(******************************************************************************
Baustein: FB_TestBase
Spezifikation: doc/Spezifikation.pdf, Kap. x.y.z
-------------------------------------------------------------------------------
erstellt:
von:
Geändert:
von:
-------------------------------------------------------------------------------
Beschreibung
Dieser Baustein stellt die Basis für einen Unittest dar und enthält
alle notwendigen Variablen und Methoden zur Testauswertung.

-------------------------------------------------------------------------------
Input
-

Output
	o_eState : EState_t;
	o_eResult: EResult_t;
******************************************************************************)
FUNCTION_BLOCK FB_Assertion
VAR_OUTPUT
    o_eState    : EAssertion_t;
    o_u32Passed : UDINT;
    o_u32Failed : UDINT;
END_VAR

(******************************************************************************
Baustein: FB_TestBase.assertFALSE
Spezifikation: doc/Spezifikation.pdf, Kap. x.y.z
-------------------------------------------------------------------------------
erstellt:
von:
Geändert:
von:
-------------------------------------------------------------------------------
Beschreibung
Diese Methode...

-------------------------------------------------------------------------------
Input
	bValue : BOOL;

Output
-
******************************************************************************)
METHOD PROTECTED FINAL _FALSE : BOOL
VAR_INPUT
	bValue : BOOL;
END_VAR

	IF bValue = FALSE THEN
		addPassed();
	ELSE
		addFailed(bFatal := FALSE);
	END_IF
END_METHOD

(******************************************************************************
Baustein: FB_TestBase.assertFALSE_Fatal
Spezifikation: doc/Spezifikation.pdf, Kap. x.y.z
-------------------------------------------------------------------------------
erstellt:
von:
Geändert:
von:
-------------------------------------------------------------------------------
Beschreibung
Diese Methode

-------------------------------------------------------------------------------
Input
	bValue : BOOL;

Output
-
******************************************************************************)
METHOD PROTECTED FINAL _FALSE_Fatal : BOOL
VAR_INPUT
	bValue : BOOL;
END_VAR

	IF bValue = FALSE THEN
		addPassed();
	ELSE
		addFailed(bFatal := true);
	END_IF
END_METHOD

(******************************************************************************
Baustein: FB_TestBase.assertTRUE
Spezifikation: doc/Spezifikation.pdf, Kap. x.y.z
-------------------------------------------------------------------------------
erstellt:
von:
Geändert:
von:
-------------------------------------------------------------------------------
Beschreibung
Diese Methode...

-------------------------------------------------------------------------------
Input
	bValue : BOOL;

Output
-
******************************************************************************)
METHOD PROTECTED FINAL _TRUE : BOOL
VAR_INPUT
	bValue : BOOL;
END_VAR

	IF bValue = true THEN
		addPassed();
	ELSE
		addFailed(bFatal := FALSE);
	END_IF
END_METHOD


(******************************************************************************
Baustein: FB_TestBase.assertTRUE_Fatal
Spezifikation: doc/Spezifikation.pdf, Kap. x.y.z
-------------------------------------------------------------------------------
erstellt:
von:
Geändert:
von:
-------------------------------------------------------------------------------
Beschreibung
Diese Methode

-------------------------------------------------------------------------------
Input
-

Output
-
******************************************************************************)
METHOD PROTECTED FINAL _TRUE_Fatal : BOOL
VAR_INPUT
	bValue : BOOL;
END_VAR

	IF bValue = TRUE THEN
		addPassed();
	ELSE
		addFailed(bFatal := true);
	END_IF
END_METHOD

METHOD INTERNAL FINAL addFailed : BOOL
VAR_INPUT
    bFatal : BOOL;
END_VAR
	
    o_u32Failed := o_u32Failed + 1;
	
	o_eState := EAssertion_t.eStateFailed;
	
	IF bFatal = true THEN
		o_eState := EAssertion_t.eStateFailedFatal;
	END_IF
END_METHOD

METHOD INTERNAL FINAL addPassed : BOOL
	
    o_u32Passed := o_u32Passed + 1;
END_METHOD

(******************************************************************************
Baustein: FB_TestBase.assertEQUAL
Spezifikation: doc/Spezifikation.pdf, Kap. x.y.z
-------------------------------------------------------------------------------
erstellt:
von:
Geändert:
von:
-------------------------------------------------------------------------------
Beschreibung
Diese Methode

-------------------------------------------------------------------------------
Input
	Actual   : ANY;
	Expected : ANY;

Output
-
******************************************************************************)
METHOD PUBLIC FINAL EQUAL : BOOL
VAR_INPUT
	Actual   : ANY;
	Expected : ANY;
END_VAR
	EQUAL := FALSE;
	
	IF validate(Actual, Expected) = FALSE THEN
		addFailed(true);
		RETURN;
	END_IF
	
	_TRUE(MEMCMP(Actual.pValue, Expected.pValue, TO_UDINT(Actual.diSize)) = 0);
END_METHOD

(******************************************************************************
Baustein: FB_TestBase.assertEQUAL_Fatal
Spezifikation: doc/Spezifikation.pdf, Kap. x.y.z
-------------------------------------------------------------------------------
erstellt:
von:
Geändert:
von:
-------------------------------------------------------------------------------
Beschreibung
Diese Methode

-------------------------------------------------------------------------------
Input
	Actual   : ANY;
	Expected : ANY;

Output
-
******************************************************************************)
METHOD PUBLIC FINAL EQUAL_Fatal : BOOL
VAR_INPUT
	Actual   : ANY;
	Expected : ANY;
END_VAR
	EQUAL_Fatal := FALSE;
	
	IF validate(Actual, Expected) = FALSE THEN
		addFailed(true);
		RETURN;
	END_IF

	_TRUE_Fatal(MEMCMP(Actual.pValue, Expected.pValue, TO_UDINT(Actual.diSize)) = 0);
END_METHOD

(******************************************************************************
Baustein: FB_TestBase.logError
Spezifikation: doc/Spezifikation.pdf, Kap. x.y.z
-------------------------------------------------------------------------------
erstellt:
von:
Geändert:
von:
-------------------------------------------------------------------------------
Beschreibung
Diese Methode

-------------------------------------------------------------------------------
Input
-

Output
-
******************************************************************************)
{attribute 'hide'} 
METHOD PROTECTED FINAL logError : BOOL
VAR_INPUT
	i_strMessage : StrMessage_t;
END_VAR

	ADSLOGSTR(msgCtrlMask 	:= ADSLOG_MSGTYPE_ERROR , 
			  msgFmtStr 	:= i_strMessage, 
			  strArg 		:= '');
END_METHOD

(******************************************************************************
Baustein: FB_TestBase.assertNotEqual
Spezifikation: doc/Spezifikation.pdf, Kap. x.y.z
-------------------------------------------------------------------------------
erstellt:
von:
Geändert:
von:
-------------------------------------------------------------------------------
Beschreibung
Diese Methode

-------------------------------------------------------------------------------
Input
	Actual   : ANY;
	Expected : ANY;

Output
-
******************************************************************************)
METHOD PUBLIC FINAL NotEqual : BOOL
VAR_INPUT
	Actual   : ANY;
	Expected : ANY;
END_VAR
	NotEqual := FALSE;
	
	IF validate(Actual, Expected) = FALSE THEN
		addFailed(true);
		RETURN;
	END_IF
	
	_TRUE(MEMCMP(Actual.pValue, Expected.pValue, TO_UDINT(Actual.diSize)) <> 0);
END_METHOD

(******************************************************************************
Baustein: FB_TestBase.assertNotEqual_Fatal
Spezifikation: doc/Spezifikation.pdf, Kap. x.y.z
-------------------------------------------------------------------------------
erstellt:
von:
Geändert:
von:
-------------------------------------------------------------------------------
Beschreibung
Diese Methode

-------------------------------------------------------------------------------
Input
	Actual   : ANY;
	Expected : ANY;

Output
-
******************************************************************************)
METHOD PUBLIC FINAL NotEqual_Fatal : BOOL
VAR_INPUT
	Actual   : ANY;
	Expected : ANY;
END_VAR
	NotEqual_Fatal := FALSE;
	
	IF validate(Actual, Expected) = FALSE THEN
		addFailed(true);
		RETURN;
	END_IF
	
	_TRUE_Fatal(MEMCMP(Actual.pValue, Expected.pValue, TO_UDINT(Actual.diSize)) <> 0);
END_METHOD

(******************************************************************************
Baustein: FB_TestBase.assertPtrEqual
Spezifikation: doc/Spezifikation.pdf, Kap. x.y.z
-------------------------------------------------------------------------------
erstellt:
von:
Geändert:
von:
-------------------------------------------------------------------------------
Beschreibung
Diese Methode

-------------------------------------------------------------------------------
Input
	pActual   : PVOID;
	pExpected : PVOID;
	
Output
-
******************************************************************************)
METHOD PUBLIC FINAL PtrEqual : BOOL
VAR_INPUT
	pActual   : PVOID;
	pExpected : PVOID;
END_VAR

	_TRUE(pActual = pExpected);
END_METHOD

(******************************************************************************
Baustein: FB_TestBase.assertPtrEqual_Fatal
Spezifikation: doc/Spezifikation.pdf, Kap. x.y.z
-------------------------------------------------------------------------------
erstellt:
von:
Geändert:
von:
-------------------------------------------------------------------------------
Beschreibung
Diese Methode

-------------------------------------------------------------------------------
Input
	pActual   : PVOID;
	pExpected : PVOID;

Output
-
******************************************************************************)
METHOD PUBLIC FINAL PtrEqual_Fatal : BOOL
VAR_INPUT
	pActual   : PVOID;
	pExpected : PVOID;
END_VAR

	_TRUE_Fatal(pActual = pExpected);
END_METHOD

(******************************************************************************
Baustein: FB_TestBase.assertPtrNotEqual
Spezifikation: doc/Spezifikation.pdf, Kap. x.y.z
-------------------------------------------------------------------------------
erstellt:
von:
Geändert:
von:
-------------------------------------------------------------------------------
Beschreibung
Diese Methode

-------------------------------------------------------------------------------
Input
	pActual   : PVOID;
	pExpected : PVOID;

Output
-
******************************************************************************)
METHOD PUBLIC FINAL PtrNotEqual : BOOL
VAR_INPUT
	pActual   : PVOID;
	pExpected : PVOID;
END_VAR

	_TRUE(pActual <> pExpected);
END_METHOD

(******************************************************************************
Baustein: FB_TestBase.assertPtrNotEqual_Fatal
Spezifikation: doc/Spezifikation.pdf, Kap. x.y.z
-------------------------------------------------------------------------------
erstellt:
von:
Geändert:
von:
-------------------------------------------------------------------------------
Beschreibung
Diese Methode

-------------------------------------------------------------------------------
Input
	pActual   : PVOID;
	pExpected : PVOID;

Output
-
******************************************************************************)
METHOD PUBLIC FINAL PtrNotEqual_Fatal : BOOL
VAR_INPUT
	pActual   : PVOID;
	pExpected : PVOID;
END_VAR

	_TRUE_Fatal(pActual <> pExpected);
END_METHOD

(******************************************************************************
Baustein: FB_TestBase.assertPtrNotNull
Spezifikation: doc/Spezifikation.pdf, Kap. x.y.z
-------------------------------------------------------------------------------
erstellt:
von:
Geändert:
von:
-------------------------------------------------------------------------------
Beschreibung
Diese Methode

-------------------------------------------------------------------------------
Input
	pActual   : PVOID;

Output
-
******************************************************************************)
METHOD PUBLIC FINAL PtrNotNull : BOOL
VAR_INPUT
	pActual   : PVOID;
END_VAR

	_TRUE(pActual <> 0);
END_METHOD

(******************************************************************************
Baustein: FB_TestBase.assertPtrNotNull_Fatal
Spezifikation: doc/Spezifikation.pdf, Kap. x.y.z
-------------------------------------------------------------------------------
erstellt:
von:
Geändert:
von:
-------------------------------------------------------------------------------
Beschreibung
Diese Methode

-------------------------------------------------------------------------------
Input
	pActual   : PVOID;

Output
-
******************************************************************************)
METHOD PUBLIC FINAL PtrNotNull_Fatal : BOOL
VAR_INPUT
	pActual   : PVOID;
END_VAR

	_TRUE_Fatal(pActual <> 0);
END_METHOD

(******************************************************************************
Baustein: FB_TestBase.assertPtrNull
Spezifikation: doc/Spezifikation.pdf, Kap. x.y.z
-------------------------------------------------------------------------------
erstellt:
von:
Geändert:
von:
-------------------------------------------------------------------------------
Beschreibung
Diese Methode

-------------------------------------------------------------------------------
Input
	pActual   : PVOID;

Output
-
******************************************************************************)
METHOD PUBLIC FINAL PtrNull : BOOL
VAR_INPUT
	pActual   : PVOID;
END_VAR

	_TRUE(pActual = 0);
END_METHOD

(******************************************************************************
Baustein: FB_TestBase.assertPtrNull_Fatal
Spezifikation: doc/Spezifikation.pdf, Kap. x.y.z
-------------------------------------------------------------------------------
erstellt:
von:
Geändert:
von:
-------------------------------------------------------------------------------
Beschreibung
Diese Methode

-------------------------------------------------------------------------------
Input
	pActual   : PVOID;

Output
-
******************************************************************************)
METHOD PUBLIC FINAL PtrNull_Fatal : BOOL
VAR_INPUT
	pActual   : PVOID;
END_VAR

	_TRUE_Fatal(pActual = 0);
END_METHOD

(******************************************************************************
Baustein: FB_TestBase.assertRealEqual
Spezifikation: doc/Spezifikation.pdf, Kap. x.y.z
-------------------------------------------------------------------------------
erstellt:
von:
Geändert:
von:
-------------------------------------------------------------------------------
Beschreibung
Diese Methode

-------------------------------------------------------------------------------
Input
	r32Actual 		: REAL;
	r32Expected 	: REAL;
	r32Granularity 	: REAL;

Output
-
******************************************************************************)
METHOD PUBLIC FINAL RealEqual : BOOL
VAR_INPUT
	r32Actual 		: REAL;
	r32Expected 	: REAL;
	r32Granularity 	: REAL;
END_VAR

	_TRUE(ABS(r32Actual-r32Expected) <= ABS(r32Granularity));
END_METHOD

(******************************************************************************
Baustein: FB_TestBase.assertRealEqual_Fatal
Spezifikation: doc/Spezifikation.pdf, Kap. x.y.z
-------------------------------------------------------------------------------
erstellt:
von:
Geändert:
von:
-------------------------------------------------------------------------------
Beschreibung
Diese Methode

-------------------------------------------------------------------------------
Input
	r32Actual 		: REAL;
	r32Expected 	: REAL;
	r32Granularity 	: REAL;

Output
-
******************************************************************************)
METHOD PUBLIC FINAL RealEqual_Fatal : BOOL
VAR_INPUT
	r32Actual 		: REAL;
	r32Expected 	: REAL;
	r32Granularity 	: REAL;
END_VAR

	_TRUE_Fatal(ABS(r32Actual-r32Expected) <= ABS(r32Granularity));
END_METHOD

(******************************************************************************
Baustein: FB_TestBase.assertRealNotEqual
Spezifikation: doc/Spezifikation.pdf, Kap. x.y.z
-------------------------------------------------------------------------------
erstellt:
von:
Geändert:
von:
-------------------------------------------------------------------------------
Beschreibung
Diese Methode

-------------------------------------------------------------------------------
Input
	r32Actual 		: REAL;
	r32Expected 	: REAL;
	r32Granularity 	: REAL;

Output
-
******************************************************************************)
METHOD PUBLIC FINAL RealNotEqual : BOOL
VAR_INPUT
	r32Actual 		: REAL;
	r32Expected 	: REAL;
	r32Granularity 	: REAL;
END_VAR

	_TRUE(ABS(r32Actual-r32Expected) > ABS(r32Granularity));
END_METHOD

(******************************************************************************
Baustein: FB_TestBase.assertRealNotEqual_Fatal
Spezifikation: doc/Spezifikation.pdf, Kap. x.y.z
-------------------------------------------------------------------------------
erstellt:
von:
Geändert:
von:
-------------------------------------------------------------------------------
Beschreibung
Diese Methode

-------------------------------------------------------------------------------
Input
	r32Actual 		: REAL;
	r32Expected 	: REAL;
	r32Granularity 	: REAL;

Output
-
******************************************************************************)
METHOD PUBLIC FINAL RealNotEqual_Fatal : BOOL
VAR_INPUT
	r32Actual 		: REAL;
	r32Expected 	: REAL;
	r32Granularity 	: REAL;
END_VAR

	_TRUE_Fatal(ABS(r32Actual-r32Expected) > ABS(r32Granularity));
END_METHOD

METHOD PUBLIC reset
VAR_INPUT
END_VAR

    o_u32Passed := o_u32Failed := 0;
    o_eState    := EAssertion_t.eStatePassed;
END_METHOD

(******************************************************************************
Baustein: FB_TestBase.assertStringEqual
Spezifikation: doc/Spezifikation.pdf, Kap. x.y.z
-------------------------------------------------------------------------------
erstellt:
von:
Geändert:
von:
-------------------------------------------------------------------------------
Beschreibung
Diese Methode

-------------------------------------------------------------------------------
Input
	pActual 	: StringHandle_t;
	pExpected 	: StringHandle_t;

Output
-
******************************************************************************)
METHOD PUBLIC FINAL StringEqual : BOOL
VAR_INPUT
	pActual 	: StringHandle_t;
	pExpected 	: StringHandle_t;
END_VAR

	IF strncmp(pActual, pExpected, LEN(pExpected^)) = TRUE THEN
		addPassed();
	ELSE
		addFailed(bFatal := FALSE);		
	END_IF
END_METHOD

(******************************************************************************
Baustein: FB_TestBase.assertStringEqual_Fatal
Spezifikation: doc/Spezifikation.pdf, Kap. x.y.z
-------------------------------------------------------------------------------
erstellt:
von:
Geändert:
von:
-------------------------------------------------------------------------------
Beschreibung
Diese Methode

-------------------------------------------------------------------------------
Input
	pActual 	: StringHandle_t;
	pExpected 	: StringHandle_t;

Output
-
******************************************************************************)
METHOD PUBLIC FINAL StringEqual_Fatal : BOOL
VAR_INPUT
	pActual 	: StringHandle_t;
	pExpected 	: StringHandle_t;
END_VAR

	IF strncmp(pActual, pExpected, LEN(pExpected^)) = TRUE THEN
		addPassed();
	ELSE
		addFailed(bFatal := TRUE);		
	END_IF
END_METHOD

(******************************************************************************
Baustein: FB_TestBase.assertStringNotEqual
Spezifikation: doc/Spezifikation.pdf, Kap. x.y.z
-------------------------------------------------------------------------------
erstellt:
von:
Geändert:
von:
-------------------------------------------------------------------------------
Beschreibung
Diese Methode

-------------------------------------------------------------------------------
Input
	pActual 	: StringHandle_t;
	pExpected 	: StringHandle_t;

Output
-
******************************************************************************)
METHOD PUBLIC FINAL StringNotEqual : BOOL
VAR_INPUT
	pActual 	: StringHandle_t;
	pExpected 	: StringHandle_t;
END_VAR

	IF strncmp(pActual, pExpected, LEN(pExpected^)) = false THEN
		addPassed();
	ELSE
		addFailed(bFatal := FALSE);		
	END_IF
END_METHOD

(******************************************************************************
Baustein: FB_TestBase.assertStringNotEqual_fatal
Spezifikation: doc/Spezifikation.pdf, Kap. x.y.z
-------------------------------------------------------------------------------
erstellt:
von:
Geändert:
von:
-------------------------------------------------------------------------------
Beschreibung
Diese Methode

-------------------------------------------------------------------------------
Input
	pExpected 	: StringHandle_t;
	pActual 	: StringHandle_t;

Output
-
******************************************************************************)
METHOD PUBLIC FINAL StringNotEqual_fatal : BOOL
VAR_INPUT
	pExpected 	: StringHandle_t;
	pActual 	: StringHandle_t;
END_VAR

	IF strncmp(pActual, pExpected, LEN(pExpected^)) = FALSE THEN
		addPassed();
	ELSE
		addFailed(bFatal := TRUE);		
	END_IF
END_METHOD

(******************************************************************************
Baustein: FB_TestBase.strncmp
Spezifikation: doc/Spezifikation.pdf, Kap. x.y.z
-------------------------------------------------------------------------------
erstellt:
von:
Geändert:
von:
-------------------------------------------------------------------------------
Beschreibung
Diese Methode

-------------------------------------------------------------------------------
Input
	strInput 	: StringHandle_t;
	strCompare 	: StringHandle_t;
	s16Size		: INT;

Output
-
******************************************************************************)
{attribute 'hide'} 
METHOD PRIVATE FINAL strncmp : BOOL
VAR_INPUT
	strInput 	: StringHandle_t;
	strCompare 	: StringHandle_t;
	s16Size		: INT;
END_VAR
VAR
	s16Size1 : INT;
	s16Size2 : INT;
	s16Diff  : INT;
END_VAR

   s16Size1:= LEN(strInput^); 
	s16Size2:= LEN(strCompare^); 
	
	strncmp := FALSE;
	
	s16Diff := s16Size1 - s16Size2;
   
	// vergleich nur wenn beide Strings
	// gleich groß sind.
	IF s16Diff  = 0 THEN

		strncmp := TRUE;
	
		WHILE(s16Size > 0) DO

			IF strInput^ <> strCompare^ THEN
				strncmp := FALSE;
			END_IF;  
 
			strInput   := strInput + 1;
			strCompare := strCompare + 1;
			s16Size    := s16Size - 1;

		END_WHILE


	
	END_IF;
END_METHOD

(******************************************************************************
Baustein: FB_TestBase.validate
Spezifikation: doc/Spezifikation.pdf, Kap. x.y.z
-------------------------------------------------------------------------------
erstellt:
von:
Geändert:
von:
-------------------------------------------------------------------------------
Beschreibung
Diese Methode

-------------------------------------------------------------------------------
Input
	var1 : ANY;
	var2 : ANY;

Output
-
******************************************************************************)
{attribute 'hide'} 
METHOD PRIVATE FINAL validate : BOOL
VAR_INPUT
	var1 : ANY;
	var2 : ANY;
END_VAR

	validate := FALSE;
	
	IF (var1.pValue = 0 OR var2.pValue = 0) THEN
		logError('Assert validation fails with NULL-Pointer');
		RETURN;
	END_IF

	IF (var1.TypeClass <> var2.TypeClass) THEN
		logError('Assert validation fails with TypeClass Error');
		RETURN;
	END_IF;	
	
	IF (var1.diSize <> var2.diSize) THEN
		logError('Assert validation fails with different size');
		RETURN;
	END_IF;	
	
	validate := true;
END_METHOD

END_FUNCTION_BLOCK

(* stored: Version 1.1.0.1, ProductVersion 3.1.4024.13
   POU FB_Assertion: Id {be4e3f75-a80c-457d-8258-79ca47381125}, SpecialFunc None
   Method _FALSE: Id {5d0cddd6-ce12-4645-b843-57f3c730a1b8}
   Method _FALSE_Fatal: Id {b16d08c0-2ccd-4f8f-9051-c40b5dce96aa}
   Method _TRUE: Id {33441899-c4bc-4d14-95fa-d19d583dc529}
   Method _TRUE_Fatal: Id {7bbdf6d0-09c5-488d-91c4-d00613f0b38a}
   Method addFailed: Id {dab15cdd-53a9-46ec-a8a6-15d74a10126c}
   Method addPassed: Id {ccf7db72-22ee-405b-b2ea-a9fe4a64ee81}
   Method EQUAL: Id {7b129b1a-521c-4e4e-b4f7-4b82ebc8b1be}
   Method EQUAL_Fatal: Id {b854c5b5-ec0c-40ad-afcf-59c63bec21fa}
   Method logError: Id {5d9700b2-77a6-4ba8-9703-51e9b1eb84d3}
   Method NotEqual: Id {9a3f38e7-93fe-476e-b34c-73ead16ddc7b}
   Method NotEqual_Fatal: Id {907fcdde-94e0-4e09-8666-32a40bdd61d1}
   Method PtrEqual: Id {0e87afe4-4cf6-4fcd-afac-72ec1b53c682}
   Method PtrEqual_Fatal: Id {cb5b95d8-041c-4e75-923c-8d0c46ecf594}
   Method PtrNotEqual: Id {d83cb42a-ec40-4298-ad3b-ca6221090345}
   Method PtrNotEqual_Fatal: Id {ccb134b1-6189-4d9b-b744-60bfe77d9e9a}
   Method PtrNotNull: Id {3f8ffc58-8d3c-432f-9dc8-a76ce2976671}
   Method PtrNotNull_Fatal: Id {9a0fc9f9-4120-43fd-9e7d-83dfc53bae0e}
   Method PtrNull: Id {0000430f-85a3-4af9-8d98-245c56d77f21}
   Method PtrNull_Fatal: Id {0ae5fe62-cb34-4a36-979d-a2dff0bba45d}
   Method RealEqual: Id {81ce98b7-bf90-4e23-98b5-2b57df1bbaa9}
   Method RealEqual_Fatal: Id {3b28ccdb-8e06-4281-b988-467260ff3e08}
   Method RealNotEqual: Id {0b529790-35ec-40e2-aba8-b5fea7f61b63}
   Method RealNotEqual_Fatal: Id {1735b76d-6f2b-4a89-998d-4bc44aedb937}
   Method reset: Id {ba2a517a-dfb4-4a68-8b79-dca5e9087525}
   Method StringEqual: Id {336b3f59-bb36-4871-b1e8-f2d66a6189bc}
   Method StringEqual_Fatal: Id {73fa3e9d-0e28-4ae5-95ea-ac67a4ef420e}
   Method StringNotEqual: Id {a5eae576-a410-4c34-ba52-60362ceb8fd0}
   Method StringNotEqual_fatal: Id {1da521b6-26f6-49ed-a3a5-439eb4c91bff}
   Method strncmp: Id {c5cf5079-398f-424e-9bbe-5c649c8eca2a}
   Method validate: Id {4963d428-7a6a-46e4-92b4-91bfe12a5c16} *)
